PROGRAM MAIN
VAR
END_VAR

END_PROGRAM

(* stored: Version 1.1.0.1
   POU MAIN: Id {c7b72bdc-d1da-4630-b0d4-6e995fa48f09} *)
